(* Logix 5000 project; controller PROJECT2 Emulate 5570 rev 30.12; software revision 30.01; part 3 of 3 *)
(* tags used below, declared in another part *)
   SIM_BNOP : BOOL;
   SIM_LevelSensor : AOI_SIMAnalogSensor_OnOff;
   SIM_ONS : BOOL;
   SIM_OutfeedSensor : AOI_SIMPartSensor;
   SIM_PowerONPB : BOOL;
   SIM_PPENABLED : BOOL;
   SIM_PTInfeedToStn1 : AOI_SIMPartTravel;
   SIM_PTStn2Fill : AOI_SIMPartTravel;
   SIM_PTStn4ToOutfeed : AOI_SIMPartTravel;
   SIM_PTStnStatus : StationStatus[20];
   SIM_PTWalkingBeam : AOI_SIMPartTravel;
   SIM_SpeedSensor : AOI_SIMAnalogSensor_OnOff;
   SIM_Stn1BottlePresentSensor : AOI_SIMPartSensor;
   SIM_Stn2BottleFilledSensor : AOI_SIMPartSensor;
   SIM_Stn2BottlePresentSensor : AOI_SIMPartSensor;
   SIM_Stn2Filler_Cylinder : AOI_SIM_2PosCyl_RsLwr;
   SIM_Stn2Filler_Fill : AOI_SIM_SimpleValve;
   SIM_Stn3BottlePresentSensor : AOI_SIMPartSensor;
   SIM_Stn3CapInsert : AOI_SIM_2PosCyl_RsLwr;
   SIM_Stn3CapPresentSensor : AOI_SIMPartSensor;
   SIM_Stn4BottlePresentSensor : AOI_SIMPartSensor;
   SIM_Stn4CapRotate : AOI_SIM_Conveyor;
   SIM_Stn4CapRotate_Cylinder : AOI_SIM_2PosCyl_RsLwr;
   SIM_WalkingBeam : AOI_SIM_3PosCyl_ExtRet;
   SIM_WalkingBeamClamp : AOI_SIM_2PosCyl_ExtRet;
   SIM_Zero : DINT;
   CapSecured : ALIAS FOR TP.PLC.YELLOW.LT;
   CH0 : ALIAS FOR Local:4:I.Ch0Data;
   CH1 : ALIAS FOR Local:4:I.Ch1Data;
   FILLSENSDELAYTIMER : TIMER;
   I2 : ALIAS FOR Local:2:I.Data;
   I31 : ALIAS FOR Ethernet3_PointIO:1:I;
   I32 : ALIAS FOR Ethernet3_PointIO:2:I;
   I33 : ALIAS FOR Ethernet3_PointIO:3:I;
   NO_OF_BOTTLES : COUNTER;
   NOOFBOT_ONESHOT3 : BOOL;
   O3 : ALIAS FOR Local:3:O.Data;
   O34 : ALIAS FOR Ethernet3_PointIO:4:O;
   O35 : ALIAS FOR Ethernet3_PointIO:5:O;
   O36 : ALIAS FOR Ethernet3_PointIO:6:O;
   TIMER : TIMER;
   TOTAL_NO_OF_BOT : DINT;
   TP : TouchPanel;
(* MainProgram, continued *)

ROUTINE R04_Walkingbeam   (* ladder *)
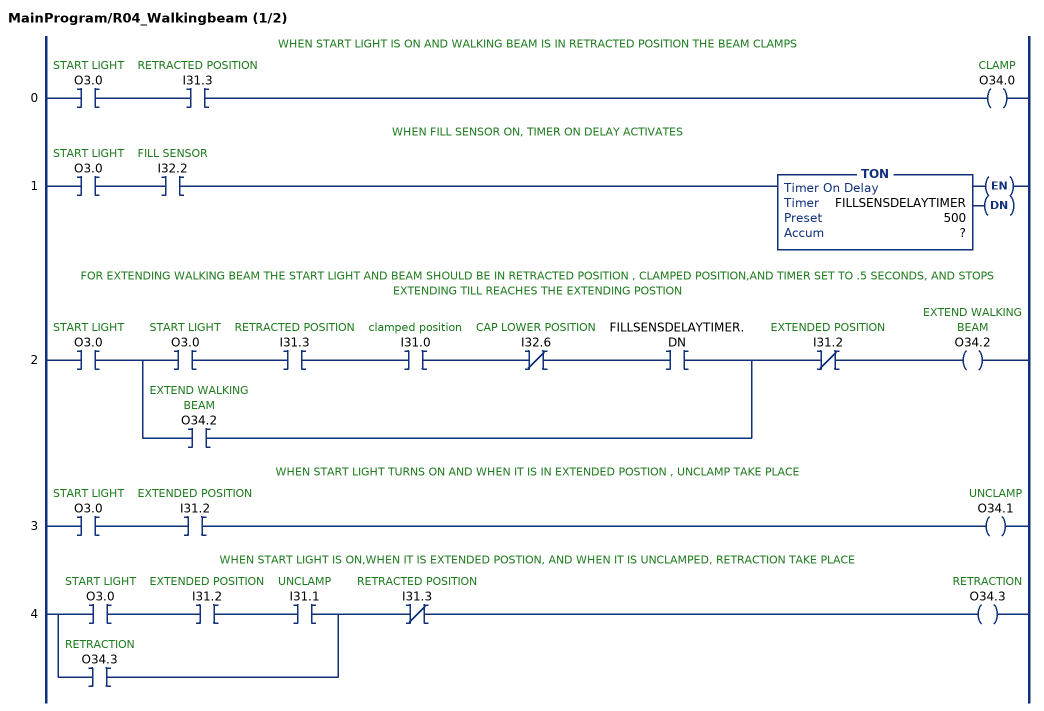
   // WHEN START LIGHT IS ON AND WALKING BEAM IS IN RETRACTED POSITION THE BEAM CLAMPS
   0: XIC(O3.0)XIC(I31.3)OTE(O34.0);
   // WHEN FILL SENSOR ON, TIMER ON DELAY ACTIVATES
   1: XIC(O3.0)XIC(I32.2)TON(FILLSENSDELAYTIMER,?,?);
   // FOR EXTENDING WALKING BEAM THE START LIGHT AND BEAM SHOULD BE IN RETRACTED POSITION , CLAMPED POSITION,AND TIMER SET TO .5 SECONDS, AND STOPS EXTENDING TILL REACHES THE EXTENDING POSTION
   2: XIC(O3.0)[XIC(O3.0) XIC(I31.3) XIC(I31.0) XIO(I32.6) XIC(FILLSENSDELAYTIMER.DN) ,XIC(O34.2) ]XIO(I31.2)OTE(O34.2);
   // WHEN START LIGHT TURNS ON AND WHEN IT IS IN EXTENDED POSTION , UNCLAMP TAKE PLACE
   3: XIC(O3.0)XIC(I31.2)OTE(O34.1);
   // WHEN START LIGHT IS ON,WHEN IT IS EXTENDED POSTION, AND WHEN IT IS UNCLAMPED, RETRACTION TAKE PLACE
   4: [XIC(O3.0) XIC(I31.2) XIC(I31.1) ,XIC(O34.3) ]XIO(I31.3)OTE(O34.3);
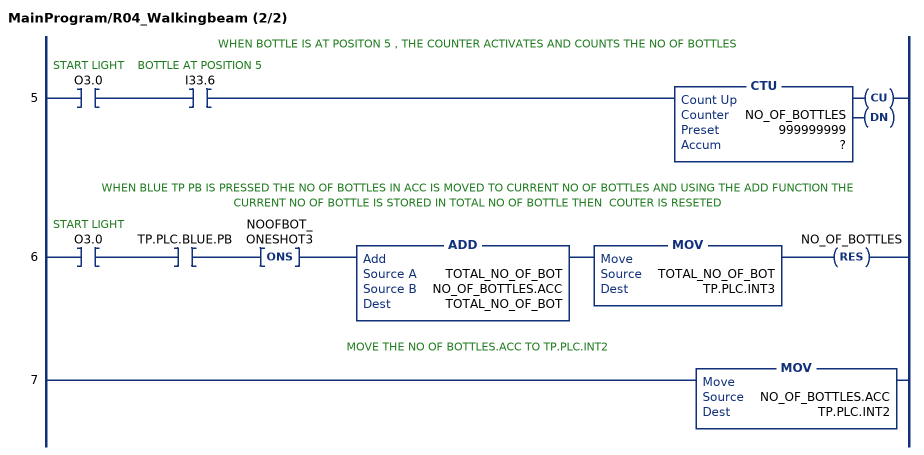
   // WHEN BOTTLE IS AT POSITON 5 , THE COUNTER ACTIVATES AND COUNTS THE NO OF BOTTLES
   5: XIC(O3.0)XIC(I33.6)CTU(NO_OF_BOTTLES,?,?);
   // WHEN BLUE TP PB IS PRESSED THE NO OF BOTTLES IN ACC IS MOVED TO CURRENT NO OF BOTTLES AND USING THE ADD FUNCTION THE CURRENT NO OF BOTTLE IS STORED IN TOTAL NO OF BOTTLE THEN  COUTER IS RESETED
   6: XIC(O3.0)XIC(TP.PLC.BLUE.PB)ONS(NOOFBOT_ONESHOT3)ADD(TOTAL_NO_OF_BOT,NO_OF_BOTTLES.ACC,TOTAL_NO_OF_BOT)MOV(TOTAL_NO_OF_BOT,TP.PLC.INT3)RES(NO_OF_BOTTLES);
   // MOVE THE NO OF BOTTLES.ACC TO TP.PLC.INT2
   7: MOV(NO_OF_BOTTLES.ACC,TP.PLC.INT2);
END_ROUTINE

ROUTINE R99_Simulate   (* ladder *)
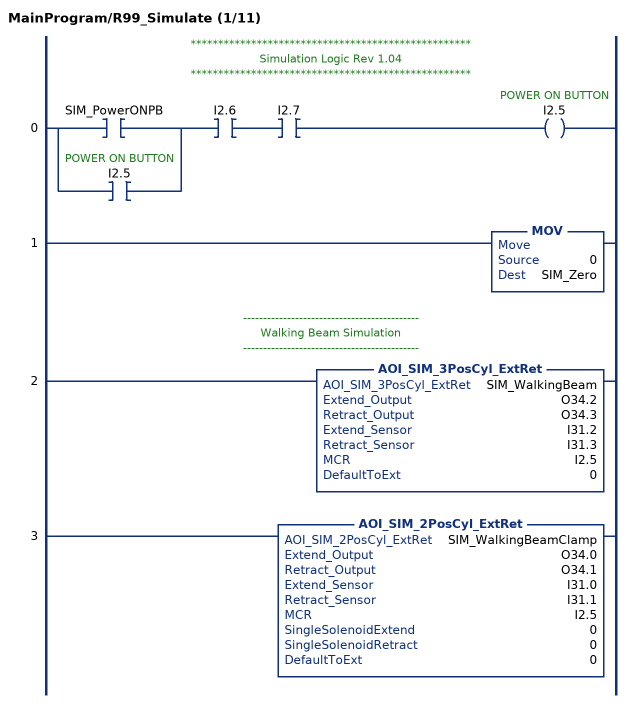
   // ***************************************************
   // Simulation Logic Rev 1.04
   // ***************************************************
   0: [XIC(SIM_PowerONPB) ,XIC(I2.5) ]XIC(I2.6)XIC(I2.7)OTE(I2.5);
   1: MOV(0,SIM_Zero);
   // --------------------------------------------
   // Walking Beam Simulation
   // --------------------------------------------
   2: AOI_SIM_3PosCyl_ExtRet(SIM_WalkingBeam,O34.2,O34.3,I31.2,I31.3,I2.5,0);
   3: AOI_SIM_2PosCyl_ExtRet(SIM_WalkingBeamClamp,O34.0,O34.1,I31.0,I31.1,I2.5,0,0,0);
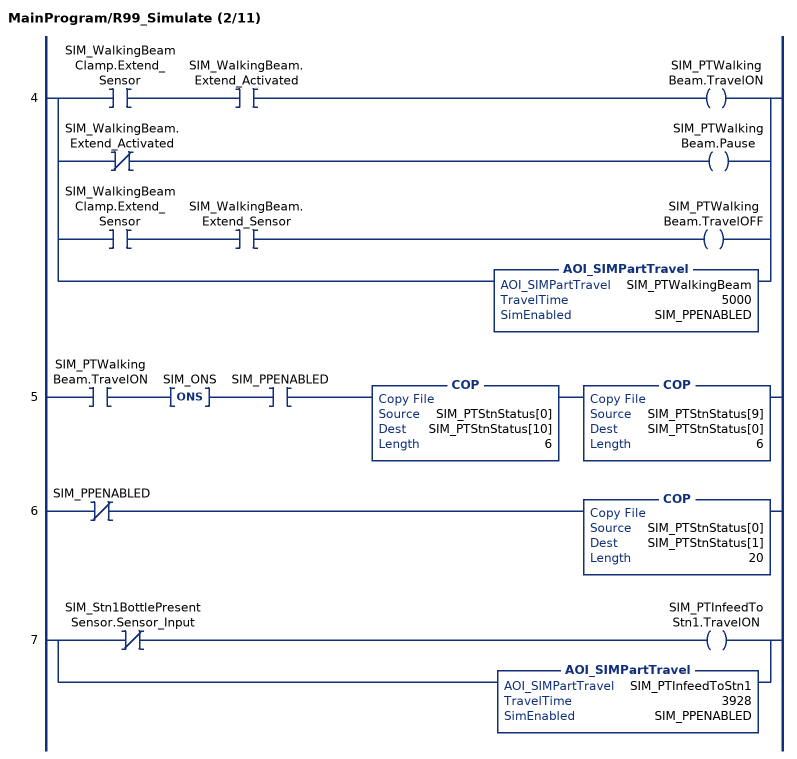
   4: [XIC(SIM_WalkingBeamClamp.Extend_Sensor) XIC(SIM_WalkingBeam.Extend_Activated) OTE(SIM_PTWalkingBeam.TravelON) ,XIO(SIM_WalkingBeam.Extend_Activated) OTE(SIM_PTWalkingBeam.Pause) ,XIC(SIM_WalkingBeamClamp.Extend_Sensor) XIC(SIM_WalkingBeam.Extend_Sensor) OTE(SIM_PTWalkingBeam.TravelOFF) ,AOI_SIMPartTravel(SIM_PTWalkingBeam,5000,SIM_PPENABLED) ];
   5: XIC(SIM_PTWalkingBeam.TravelON)ONS(SIM_ONS)XIC(SIM_PPENABLED)COP(SIM_PTStnStatus[0],SIM_PTStnStatus[10],6)COP(SIM_PTStnStatus[9],SIM_PTStnStatus[0],6);
   6: XIO(SIM_PPENABLED)COP(SIM_PTStnStatus[0],SIM_PTStnStatus[1],20);
   7: [XIO(SIM_Stn1BottlePresentSensor.Sensor_Input) OTE(SIM_PTInfeedToStn1.TravelON) ,AOI_SIMPartTravel(SIM_PTInfeedToStn1,3928,SIM_PPENABLED) ];
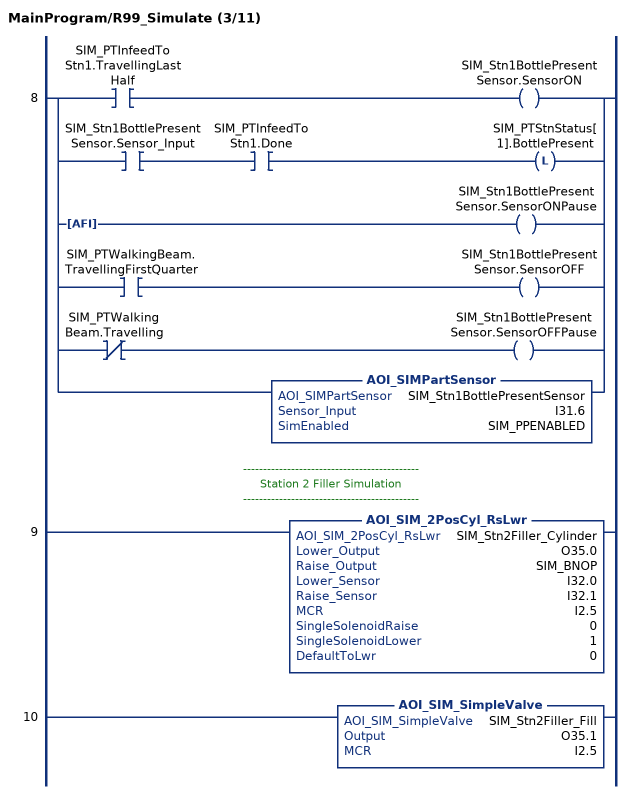
   8: [XIC(SIM_PTInfeedToStn1.TravellingLastHalf) OTE(SIM_Stn1BottlePresentSensor.SensorON) ,XIC(SIM_Stn1BottlePresentSensor.Sensor_Input) XIC(SIM_PTInfeedToStn1.Done) OTL(SIM_PTStnStatus[1].BottlePresent) ,AFI() OTE(SIM_Stn1BottlePresentSensor.SensorONPause) ,XIC(SIM_PTWalkingBeam.TravellingFirstQuarter) OTE(SIM_Stn1BottlePresentSensor.SensorOFF) ,XIO(SIM_PTWalkingBeam.Travelling) OTE(SIM_Stn1BottlePresentSensor.SensorOFFPause) ,AOI_SIMPartSensor(SIM_Stn1BottlePresentSensor,I31.6,SIM_PPENABLED) ];
   // --------------------------------------------
   // Station 2 Filler Simulation
   // --------------------------------------------
   9: AOI_SIM_2PosCyl_RsLwr(SIM_Stn2Filler_Cylinder,O35.0,SIM_BNOP,I32.0,I32.1,I2.5,0,1,0);
   10: AOI_SIM_SimpleValve(SIM_Stn2Filler_Fill,O35.1,I2.5);
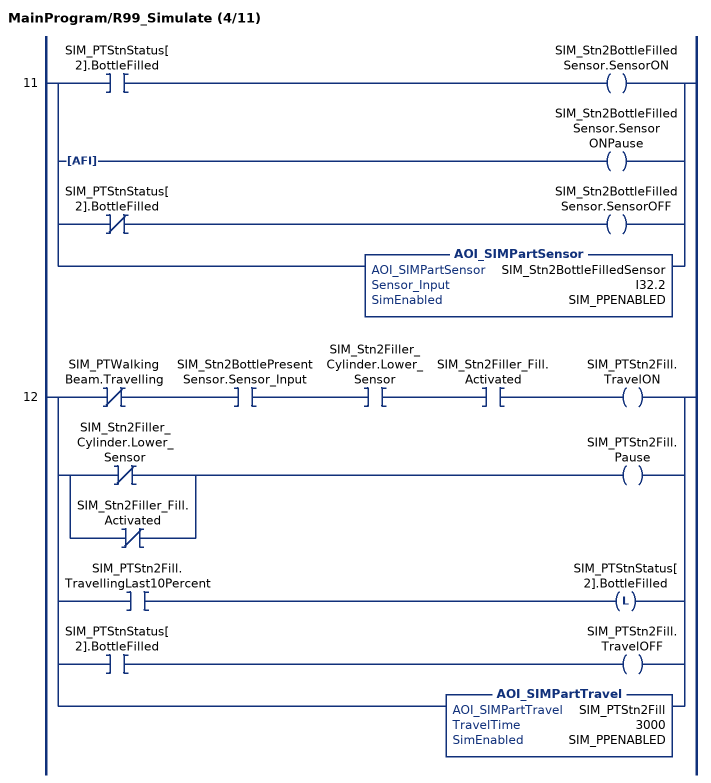
   11: [XIC(SIM_PTStnStatus[2].BottleFilled) OTE(SIM_Stn2BottleFilledSensor.SensorON) ,AFI() OTE(SIM_Stn2BottleFilledSensor.SensorONPause) ,XIO(SIM_PTStnStatus[2].BottleFilled) OTE(SIM_Stn2BottleFilledSensor.SensorOFF) ,AOI_SIMPartSensor(SIM_Stn2BottleFilledSensor,I32.2,SIM_PPENABLED) ];
   12: [XIO(SIM_PTWalkingBeam.Travelling) XIC(SIM_Stn2BottlePresentSensor.Sensor_Input) XIC(SIM_Stn2Filler_Cylinder.Lower_Sensor) XIC(SIM_Stn2Filler_Fill.Activated) OTE(SIM_PTStn2Fill.TravelON) ,[XIO(SIM_Stn2Filler_Cylinder.Lower_Sensor) ,XIO(SIM_Stn2Filler_Fill.Activated) ] OTE(SIM_PTStn2Fill.Pause) ,XIC(SIM_PTStn2Fill.TravellingLast10Percent) OTL(SIM_PTStnStatus[2].BottleFilled) ,XIC(SIM_PTStnStatus[2].BottleFilled) OTE(SIM_PTStn2Fill.TravelOFF) ,AOI_SIMPartTravel(SIM_PTStn2Fill,3000,SIM_PPENABLED) ];
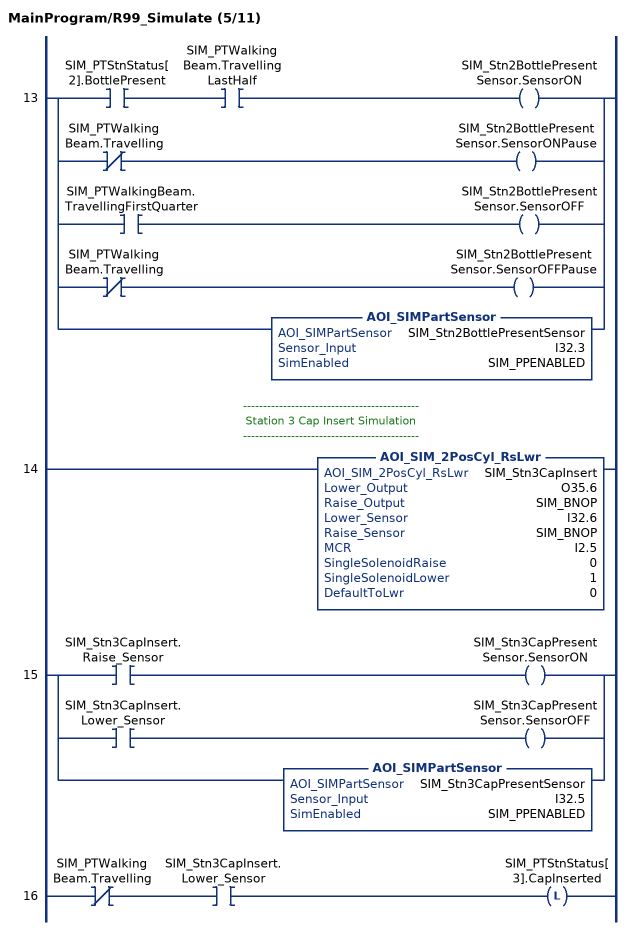
   13: [XIC(SIM_PTStnStatus[2].BottlePresent) XIC(SIM_PTWalkingBeam.TravellingLastHalf) OTE(SIM_Stn2BottlePresentSensor.SensorON) ,XIO(SIM_PTWalkingBeam.Travelling) OTE(SIM_Stn2BottlePresentSensor.SensorONPause) ,XIC(SIM_PTWalkingBeam.TravellingFirstQuarter) OTE(SIM_Stn2BottlePresentSensor.SensorOFF) ,XIO(SIM_PTWalkingBeam.Travelling) OTE(SIM_Stn2BottlePresentSensor.SensorOFFPause) ,AOI_SIMPartSensor(SIM_Stn2BottlePresentSensor,I32.3,SIM_PPENABLED) ];
   // --------------------------------------------
   // Station 3 Cap Insert Simulation
   // --------------------------------------------
   14: AOI_SIM_2PosCyl_RsLwr(SIM_Stn3CapInsert,O35.6,SIM_BNOP,I32.6,SIM_BNOP,I2.5,0,1,0);
   15: [XIC(SIM_Stn3CapInsert.Raise_Sensor) OTE(SIM_Stn3CapPresentSensor.SensorON) ,XIC(SIM_Stn3CapInsert.Lower_Sensor) OTE(SIM_Stn3CapPresentSensor.SensorOFF) ,AOI_SIMPartSensor(SIM_Stn3CapPresentSensor,I32.5,SIM_PPENABLED) ];
   16: XIO(SIM_PTWalkingBeam.Travelling)XIC(SIM_Stn3CapInsert.Lower_Sensor)OTL(SIM_PTStnStatus[3].CapInserted);
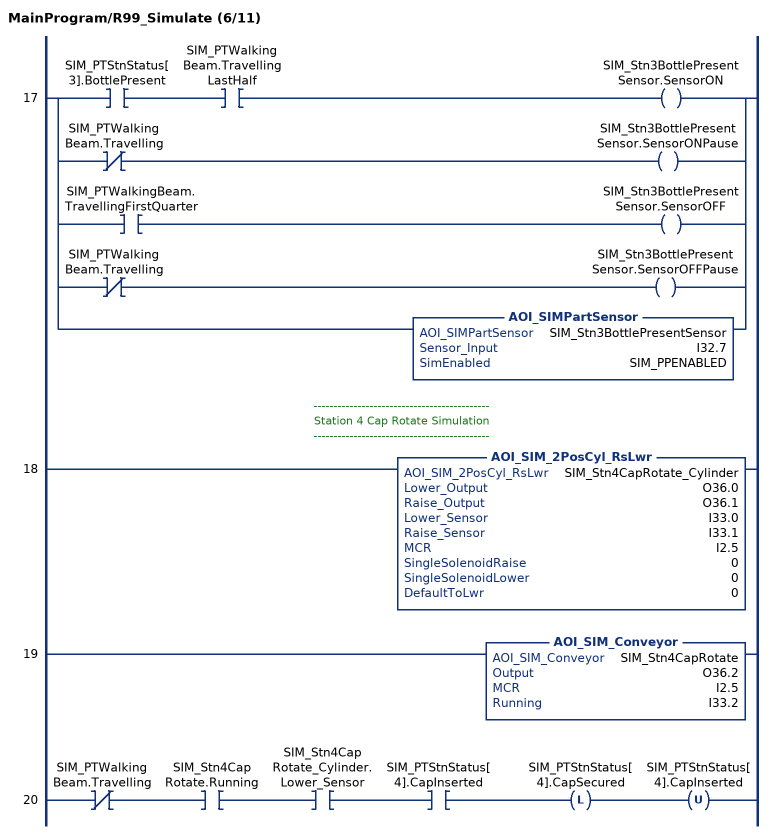
   17: [XIC(SIM_PTStnStatus[3].BottlePresent) XIC(SIM_PTWalkingBeam.TravellingLastHalf) OTE(SIM_Stn3BottlePresentSensor.SensorON) ,XIO(SIM_PTWalkingBeam.Travelling) OTE(SIM_Stn3BottlePresentSensor.SensorONPause) ,XIC(SIM_PTWalkingBeam.TravellingFirstQuarter) OTE(SIM_Stn3BottlePresentSensor.SensorOFF) ,XIO(SIM_PTWalkingBeam.Travelling) OTE(SIM_Stn3BottlePresentSensor.SensorOFFPause) ,AOI_SIMPartSensor(SIM_Stn3BottlePresentSensor,I32.7,SIM_PPENABLED) ];
   // --------------------------------------------
   // Station 4 Cap Rotate Simulation
   // --------------------------------------------
   18: AOI_SIM_2PosCyl_RsLwr(SIM_Stn4CapRotate_Cylinder,O36.0,O36.1,I33.0,I33.1,I2.5,0,0,0);
   19: AOI_SIM_Conveyor(SIM_Stn4CapRotate,O36.2,I2.5,I33.2);
   20: XIO(SIM_PTWalkingBeam.Travelling)XIC(SIM_Stn4CapRotate.Running)XIC(SIM_Stn4CapRotate_Cylinder.Lower_Sensor)XIC(SIM_PTStnStatus[4].CapInserted)OTL(SIM_PTStnStatus[4].CapSecured)OTU(SIM_PTStnStatus[4].CapInserted);
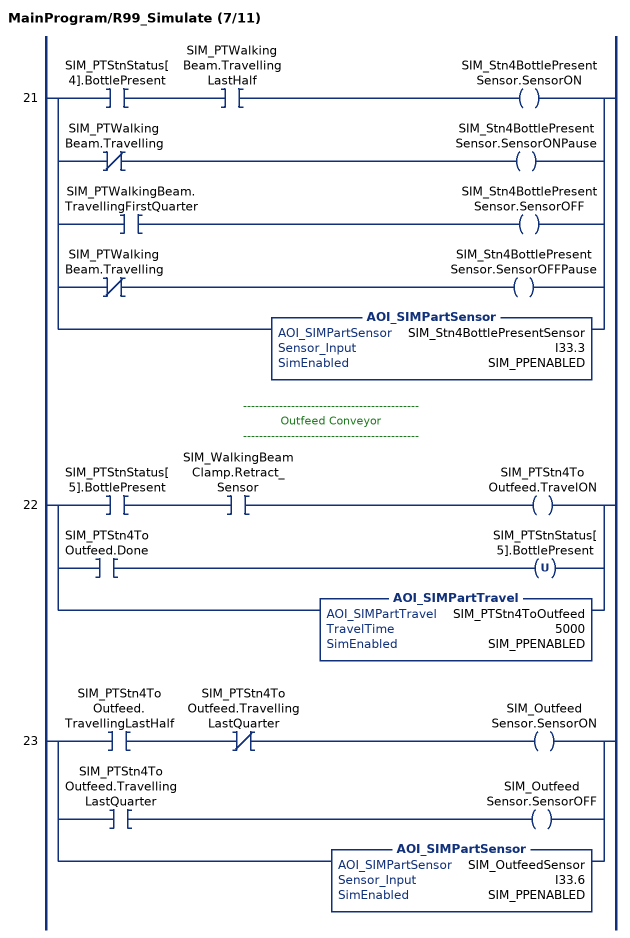
   21: [XIC(SIM_PTStnStatus[4].BottlePresent) XIC(SIM_PTWalkingBeam.TravellingLastHalf) OTE(SIM_Stn4BottlePresentSensor.SensorON) ,XIO(SIM_PTWalkingBeam.Travelling) OTE(SIM_Stn4BottlePresentSensor.SensorONPause) ,XIC(SIM_PTWalkingBeam.TravellingFirstQuarter) OTE(SIM_Stn4BottlePresentSensor.SensorOFF) ,XIO(SIM_PTWalkingBeam.Travelling) OTE(SIM_Stn4BottlePresentSensor.SensorOFFPause) ,AOI_SIMPartSensor(SIM_Stn4BottlePresentSensor,I33.3,SIM_PPENABLED) ];
   // --------------------------------------------
   // Outfeed Conveyor
   // --------------------------------------------
   22: [XIC(SIM_PTStnStatus[5].BottlePresent) XIC(SIM_WalkingBeamClamp.Retract_Sensor) OTE(SIM_PTStn4ToOutfeed.TravelON) ,XIC(SIM_PTStn4ToOutfeed.Done) OTU(SIM_PTStnStatus[5].BottlePresent) ,AOI_SIMPartTravel(SIM_PTStn4ToOutfeed,5000,SIM_PPENABLED) ];
   23: [XIC(SIM_PTStn4ToOutfeed.TravellingLastHalf) XIO(SIM_PTStn4ToOutfeed.TravellingLastQuarter) OTE(SIM_OutfeedSensor.SensorON) ,XIC(SIM_PTStn4ToOutfeed.TravellingLastQuarter) OTE(SIM_OutfeedSensor.SensorOFF) ,AOI_SIMPartSensor(SIM_OutfeedSensor,I33.6,SIM_PPENABLED) ];
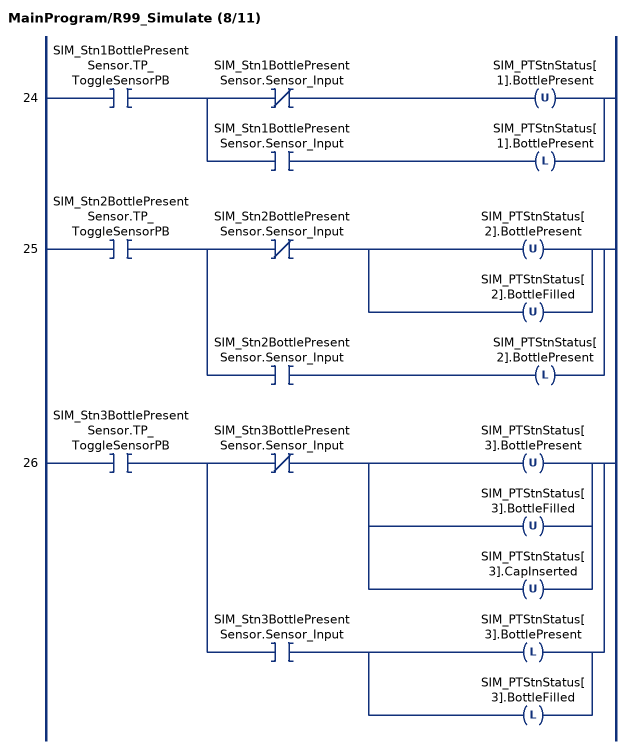
   24: XIC(SIM_Stn1BottlePresentSensor.TP_ToggleSensorPB)[XIO(SIM_Stn1BottlePresentSensor.Sensor_Input) OTU(SIM_PTStnStatus[1].BottlePresent) ,XIC(SIM_Stn1BottlePresentSensor.Sensor_Input) OTL(SIM_PTStnStatus[1].BottlePresent) ];
   25: XIC(SIM_Stn2BottlePresentSensor.TP_ToggleSensorPB)[XIO(SIM_Stn2BottlePresentSensor.Sensor_Input) [OTU(SIM_PTStnStatus[2].BottlePresent) ,OTU(SIM_PTStnStatus[2].BottleFilled) ] ,XIC(SIM_Stn2BottlePresentSensor.Sensor_Input) OTL(SIM_PTStnStatus[2].BottlePresent) ];
   26: XIC(SIM_Stn3BottlePresentSensor.TP_ToggleSensorPB)[XIO(SIM_Stn3BottlePresentSensor.Sensor_Input) [OTU(SIM_PTStnStatus[3].BottlePresent) ,OTU(SIM_PTStnStatus[3].BottleFilled) ,OTU(SIM_PTStnStatus[3].CapInserted) ] ,XIC(SIM_Stn3BottlePresentSensor.Sensor_Input) [OTL(SIM_PTStnStatus[3].BottlePresent) ,OTL(SIM_PTStnStatus[3].BottleFilled) ] ];
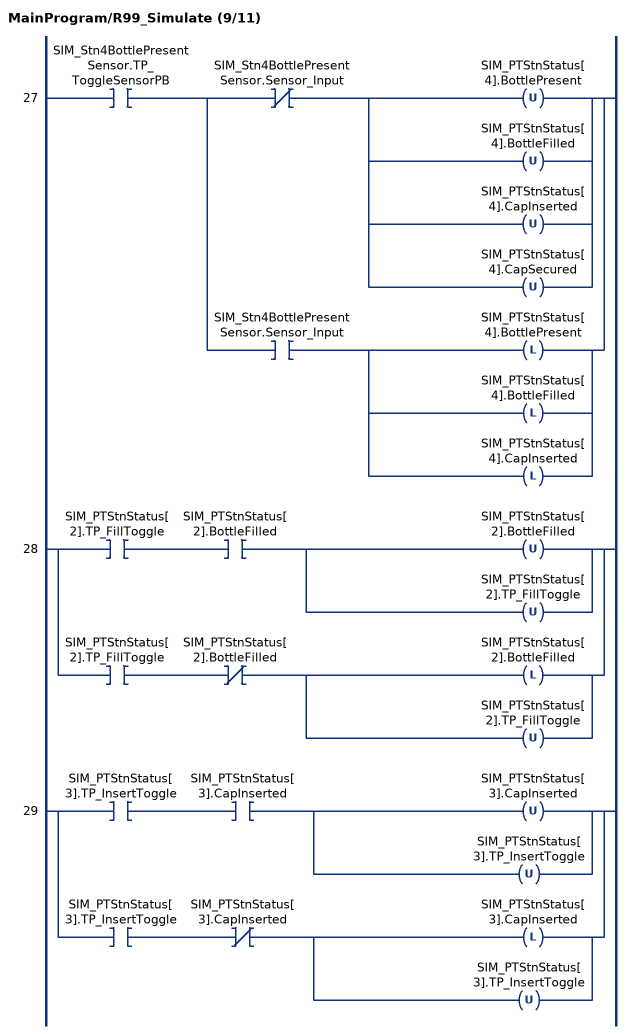
   27: XIC(SIM_Stn4BottlePresentSensor.TP_ToggleSensorPB)[XIO(SIM_Stn4BottlePresentSensor.Sensor_Input) [OTU(SIM_PTStnStatus[4].BottlePresent) ,OTU(SIM_PTStnStatus[4].BottleFilled) ,OTU(SIM_PTStnStatus[4].CapInserted) ,OTU(SIM_PTStnStatus[4].CapSecured) ] ,XIC(SIM_Stn4BottlePresentSensor.Sensor_Input) [OTL(SIM_PTStnStatus[4].BottlePresent) ,OTL(SIM_PTStnStatus[4].BottleFilled) ,OTL(SIM_PTStnStatus[4].CapInserted) ] ];
   28: [XIC(SIM_PTStnStatus[2].TP_FillToggle) XIC(SIM_PTStnStatus[2].BottleFilled) [OTU(SIM_PTStnStatus[2].BottleFilled) ,OTU(SIM_PTStnStatus[2].TP_FillToggle) ] ,XIC(SIM_PTStnStatus[2].TP_FillToggle) XIO(SIM_PTStnStatus[2].BottleFilled) [OTL(SIM_PTStnStatus[2].BottleFilled) ,OTU(SIM_PTStnStatus[2].TP_FillToggle) ] ];
   29: [XIC(SIM_PTStnStatus[3].TP_InsertToggle) XIC(SIM_PTStnStatus[3].CapInserted) [OTU(SIM_PTStnStatus[3].CapInserted) ,OTU(SIM_PTStnStatus[3].TP_InsertToggle) ] ,XIC(SIM_PTStnStatus[3].TP_InsertToggle) XIO(SIM_PTStnStatus[3].CapInserted) [OTL(SIM_PTStnStatus[3].CapInserted) ,OTU(SIM_PTStnStatus[3].TP_InsertToggle) ] ];
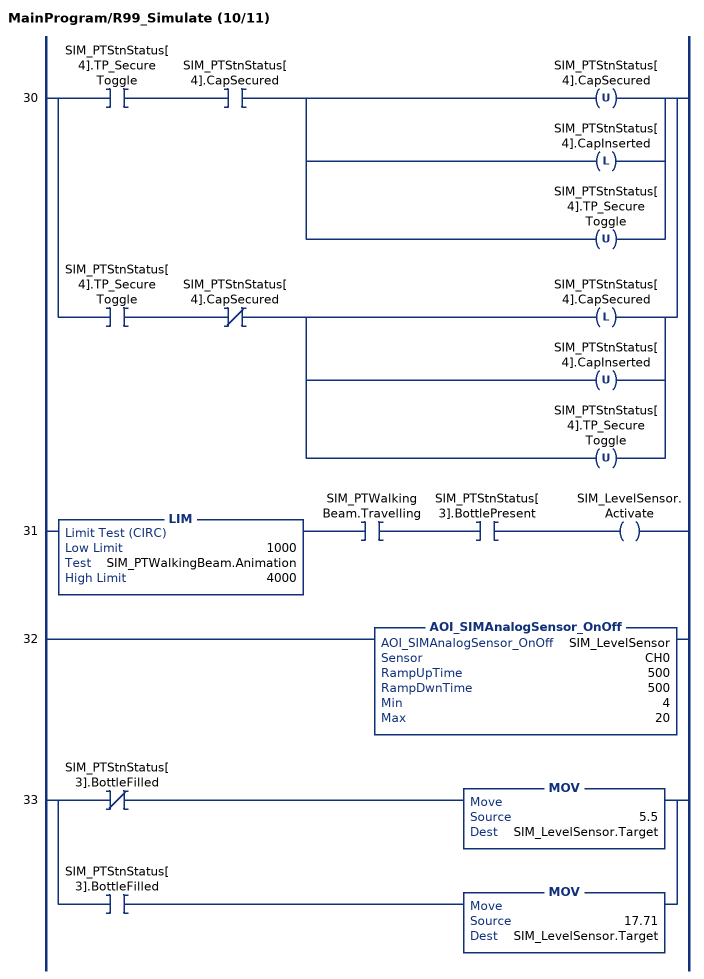
   30: [XIC(SIM_PTStnStatus[4].TP_SecureToggle) XIC(SIM_PTStnStatus[4].CapSecured) [OTU(SIM_PTStnStatus[4].CapSecured) ,OTL(SIM_PTStnStatus[4].CapInserted) ,OTU(SIM_PTStnStatus[4].TP_SecureToggle) ] ,XIC(SIM_PTStnStatus[4].TP_SecureToggle) XIO(SIM_PTStnStatus[4].CapSecured) [OTL(SIM_PTStnStatus[4].CapSecured) ,OTU(SIM_PTStnStatus[4].CapInserted) ,OTU(SIM_PTStnStatus[4].TP_SecureToggle) ] ];
   31: LIM(1000,SIM_PTWalkingBeam.Animation,4000)XIC(SIM_PTWalkingBeam.Travelling)XIC(SIM_PTStnStatus[3].BottlePresent)OTE(SIM_LevelSensor.Activate);
   32: AOI_SIMAnalogSensor_OnOff(SIM_LevelSensor,CH0,500,500,4,20);
   33: [XIO(SIM_PTStnStatus[3].BottleFilled) MOV(5.5,SIM_LevelSensor.Target) ,XIC(SIM_PTStnStatus[3].BottleFilled) MOV(17.71,SIM_LevelSensor.Target) ];
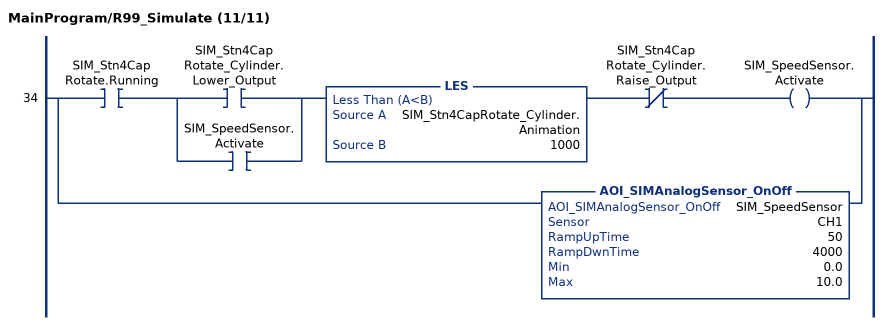
   34: [XIC(SIM_Stn4CapRotate.Running) [XIC(SIM_Stn4CapRotate_Cylinder.Lower_Output) ,XIC(SIM_SpeedSensor.Activate) ] LES(SIM_Stn4CapRotate_Cylinder.Animation,1000) XIO(SIM_Stn4CapRotate_Cylinder.Raise_Output) OTE(SIM_SpeedSensor.Activate) ,AOI_SIMAnalogSensor_OnOff(SIM_SpeedSensor,CH1,50,4000,0.0,10.0) ];
END_ROUTINE
END_PROGRAM
